// Mitsubishi GX Works2 project: MitTestPython   PLC: Q10UDEH

PROGRAM MAIN
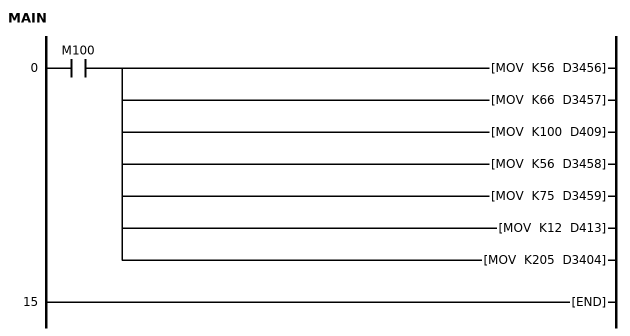
0     LD      M100
      MOV     K56 D3456
      MOV     K66 D3457
      MOV     K100 D409
      MOV     K56 D3458
      MOV     K75 D3459
      MOV     K12 D413
      MOV     K205 D3404
15    END
END_PROGRAM

// device comments not shown above
X21  ; READ
Y105A  ; OK TO   READ
M99  ; TEST
